PROGRAM MAIN
VAR
END_VAR

END_PROGRAM

(* stored: Version 1.1.0.1
   POU MAIN: Id {d4fdf5aa-2f90-41e9-a924-7e93eef6c38a} *)
